# EPICS IOC start-up script: examples/test/PSI/ep3744.iocsh
#- mXsXXX naming
require ecmccfg, "NAMING=mXsXXX"

#- add slaves
${SCRIPTEXEC} ${ecmccfg_DIR}addSlave.cmd, "HW_DESC=EP3744, SLAVE_ID=1"
ecmcConfigOrDie "Cfg.EcAddSdo(${ECMC_EC_SLAVE_NUM},0x8020,0x19,7,2)"
